PROGRAM MAIN_TEST
VAR
  FileMemoryTest: FileMemory_Test;
END_VAR

GVL_EventLogger.runner();
TcUnit.RUN();

END_PROGRAM

(* stored: Version 1.1.0.1, ProductVersion 3.1.4024.6
   POU MAIN_TEST: Id {c5a022a8-f196-47f6-9c7f-1db1bc1f3d17}, SpecialFunc None *)
